// TIA Portal V19 export
FUNCTION "Utgangskretser" : Void   // FC3, LAD
{ S7_Optimized_Access := 'TRUE' }
// stored: SetENOAutomatically false
BEGIN

REGION Network 1
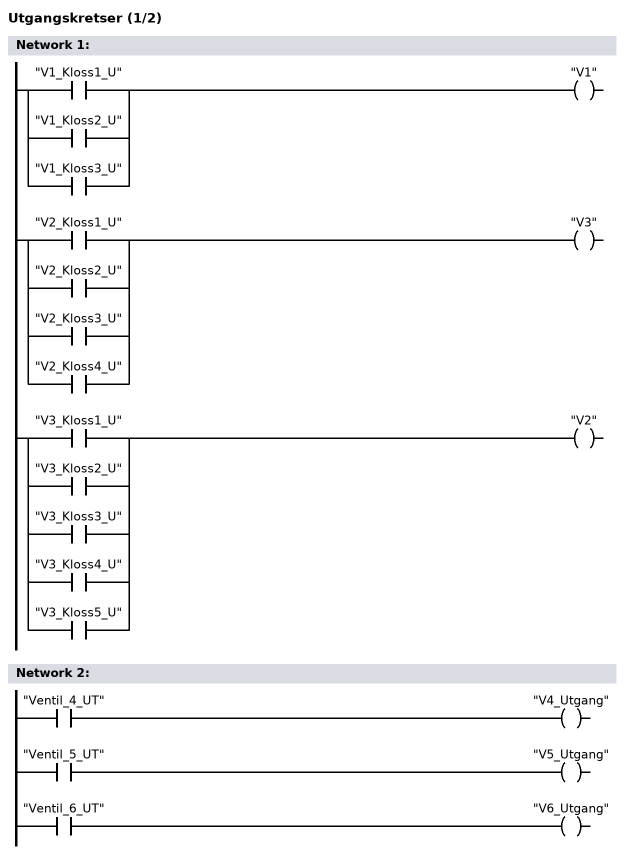
   RUNG wire#powerrail
      Contact( "V1_Kloss1_U" )
      wire#w1
      Coil( "V1" )
   END_RUNG
   RUNG wire#powerrail
      Contact( "V1_Kloss2_U" )
   END_RUNG wire#w1
   RUNG wire#powerrail
      Contact( "V1_Kloss3_U" )
   END_RUNG wire#w1
   RUNG wire#powerrail
      Contact( "V2_Kloss1_U" )
      wire#w2
      Coil( "V3" )
   END_RUNG
   RUNG wire#powerrail
      Contact( "V2_Kloss2_U" )
   END_RUNG wire#w2
   RUNG wire#powerrail
      Contact( "V2_Kloss3_U" )
   END_RUNG wire#w2
   RUNG wire#powerrail
      Contact( "V2_Kloss4_U" )
   END_RUNG wire#w2
   RUNG wire#powerrail
      Contact( "V3_Kloss1_U" )
      wire#w3
      Coil( "V2" )
   END_RUNG
   RUNG wire#powerrail
      Contact( "V3_Kloss2_U" )
   END_RUNG wire#w3
   RUNG wire#powerrail
      Contact( "V3_Kloss3_U" )
   END_RUNG wire#w3
   RUNG wire#powerrail
      Contact( "V3_Kloss4_U" )
   END_RUNG wire#w3
   RUNG wire#powerrail
      Contact( "V3_Kloss5_U" )
   END_RUNG wire#w3
   // the same network as SCL:
   "V1" := "V1_Kloss1_U" OR "V1_Kloss2_U" OR "V1_Kloss3_U";
   "V3" := "V2_Kloss1_U" OR "V2_Kloss2_U" OR "V2_Kloss3_U" OR "V2_Kloss4_U";
   "V2" := "V3_Kloss1_U" OR "V3_Kloss2_U" OR "V3_Kloss3_U" OR "V3_Kloss4_U" OR "V3_Kloss5_U";
END_REGION

REGION Network 2
   RUNG wire#powerrail
      Contact( "Ventil_4_UT" )
      Coil( "V4_Utgang" )
   END_RUNG
   RUNG wire#powerrail
      Contact( "Ventil_5_UT" )
      Coil( "V5_Utgang" )
   END_RUNG
   RUNG wire#powerrail
      Contact( "Ventil_6_UT" )
      Coil( "V6_Utgang" )
   END_RUNG
   // the same network as SCL:
   "V4_Utgang" := "Ventil_4_UT";
   "V5_Utgang" := "Ventil_5_UT";
   "V6_Utgang" := "Ventil_6_UT";
END_REGION

REGION Network 3
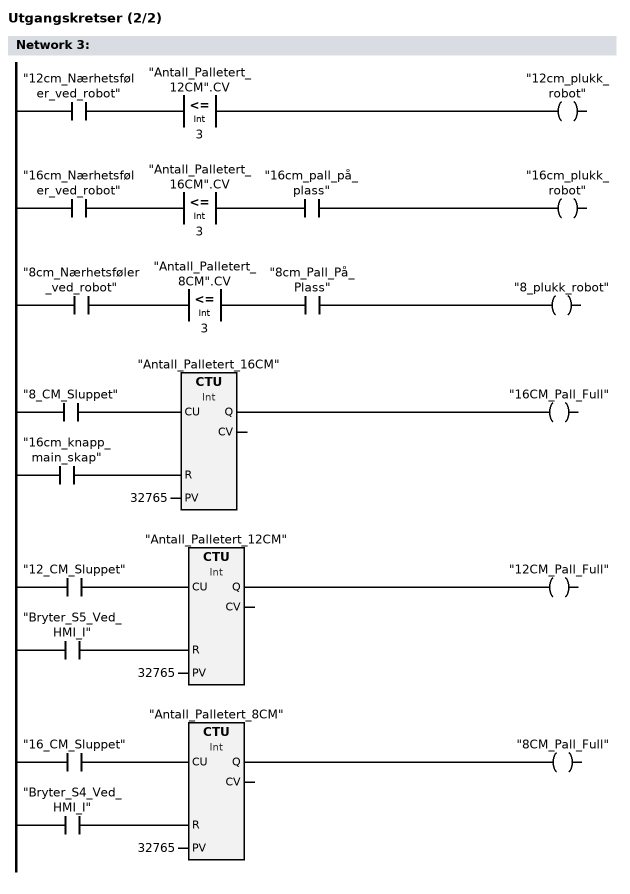
   RUNG wire#powerrail
      Contact( "12cm_Nærhetsføler_ved_robot" )
      { S7_Templates := "SrcType := Int" } LE_Contact(in1 := "Antall_Palletert_12CM".CV, in2 := 3)
      Coil( "12cm_plukk_robot" )
   END_RUNG
   RUNG wire#powerrail
      Contact( "16cm_Nærhetsføler_ved_robot" )
      { S7_Templates := "SrcType := Int" } LE_Contact(in1 := "Antall_Palletert_16CM".CV, in2 := 3)
      Contact( "16cm_pall_på_plass" )
      Coil( "16cm_plukk_robot" )
   END_RUNG
   RUNG wire#powerrail
      Contact( "8cm_Nærhetsføler_ved_robot" )
      { S7_Templates := "SrcType := Int" } LE_Contact(in1 := "Antall_Palletert_8CM".CV, in2 := 3)
      Contact( "8cm_Pall_På_Plass" )
      Coil( "8_plukk_robot" )
   END_RUNG
   RUNG wire#powerrail
      Contact( "8_CM_Sluppet" )
      { S7_Templates := "value_type := Int" } "Antall_Palletert_16CM".CTU(r := wire#w1, pv := 32765, cv =>)
      Coil( "16CM_Pall_Full" )
   END_RUNG
   RUNG wire#powerrail
      Contact( "16cm_knapp_main_skap" )
   END_RUNG wire#w1
   RUNG wire#powerrail
      Contact( "12_CM_Sluppet" )
      { S7_Templates := "value_type := Int" } "Antall_Palletert_12CM".CTU(r := wire#w2, pv := 32765, cv =>)
      Coil( "12CM_Pall_Full" )
   END_RUNG
   RUNG wire#powerrail
      Contact( "Bryter_S5_Ved_HMI_I" )
   END_RUNG wire#w2
   RUNG wire#powerrail
      Contact( "16_CM_Sluppet" )
      { S7_Templates := "value_type := Int" } "Antall_Palletert_8CM".CTU(r := wire#w3, pv := 32765, cv =>)
      Coil( "8CM_Pall_Full" )
   END_RUNG
   RUNG wire#powerrail
      Contact( "Bryter_S4_Ved_HMI_I" )
   END_RUNG wire#w3
   // the same network as SCL:
   "12cm_plukk_robot" := "12cm_Nærhetsføler_ved_robot" AND ("Antall_Palletert_12CM".CV <= 3);
   "16cm_plukk_robot" := "16cm_Nærhetsføler_ved_robot" AND ("Antall_Palletert_16CM".CV <= 3) AND "16cm_pall_på_plass";
   "8_plukk_robot" := "8cm_Nærhetsføler_ved_robot" AND ("Antall_Palletert_8CM".CV <= 3) AND "8cm_Pall_På_Plass";
   "Antall_Palletert_16CM".CTU(CU := "8_CM_Sluppet", R := "16cm_knapp_main_skap", PV := 32765);
   "16CM_Pall_Full" := "Antall_Palletert_16CM".Q;
   "Antall_Palletert_12CM".CTU(CU := "12_CM_Sluppet", R := "Bryter_S5_Ved_HMI_I", PV := 32765);
   "12CM_Pall_Full" := "Antall_Palletert_12CM".Q;
   "Antall_Palletert_8CM".CTU(CU := "16_CM_Sluppet", R := "Bryter_S4_Ved_HMI_I", PV := 32765);
   "8CM_Pall_Full" := "Antall_Palletert_8CM".Q;
END_REGION
END_FUNCTION
